Universal Robots PolyScope program: sockets.urp

Program sockets (installation=default directory=/programs/Alumnes/Lua/socketsTestV1 createdIn=5.17.3 lastSavedIn=5.20.0 robotSerialNumber=20205300829)
Calibrated DH parameters: a=[0.000012, -0.242852, -0.179835, 0.000093, -0.000124, 0]; d=[0.151981, 5.088974, 36.181125, -41.139477, 0.085414, 0.092081]; alpha=[1.572112, -0.003585, 0.002783, 1.571586, -1.572466, 0]; deltaTheta=[0, -0.074993, 0.643315, -0.56833, 0.000002, 0]
InitVariablesNode
BeforeStart
  socketTxt := "s1"
  len := 2
  Script file /programs/Alumnes/Lua/socketsTestV1/functions.script
    | def operacio(mode, currentWidht):
    | 	socket_send_byte(mode ,socketTxt)
    | 	socket_send_byte(currentWidht, socketTxt)
    | 	return socket_read_byte_list(len, socketTxt, 2)
    | end
    | 
    | def open(data, targetWidht):
    | 	currentWidht=data[2]
    | 	while(currentWidht<targetWidht):
    | 		data=operacio(1, currentWidht)
    | 		currentWidht=data[2]
    | 	end
    | 	data=operacio(0, currentWidht)
    | 	return data
    | end
    | 
    | def close(data, targetWidht):
    | 	currentWidht=data[2]
    | 	while(currentWidht>targetWidht):
    | 		data=operacio(2, currentWidht)
    | 		currentWidht=data[2]
    | 	end
    | 	data=operacio(0, currentWidht)
    | 	return data
    | end
  initial_pose := get_actual_tcp_pose()
  ip := "172.30.3.149"
  socket := False
Robot Program (runOnlyOnce=false)
  Loop While (checkContinuously=false) expression=socket≟False
    socket := socket_open(ip, 8080,"s1")
  data := socket_read_byte_list(2, "s1", 4)
  Popup Error (haltProgram=false inputType=Variable) variable=data
  Loop While (checkContinuously=false) expression=True
    SuppressedNode
      Script: operacio(2, 45)
    data := close(data,25)
    data := open(data, 42)
